(* IEC 61131-3 sources: learning-path/05_oop_in_st/exercises/2_interfaces/src, 2 files *)

(* ---- basicTank.st ---- *)
NAMESPACE FluidHandlingClass

    //Update the class to implement the Interface
    class Tank
        VAR PUBLIC
            inletValve: ValveClass;
            outletValve: ValveClass;
        END_VAR

        METHOD PRIVATE OpenInlet
            inletValve.Open();
        END_METHOD
        METHOD PRIVATE OpenOutlet
            outletValve.Open();
        END_METHOD
        METHOD PRIVATE CloseInlet
            inletValve.Close();
        END_METHOD
        METHOD PRIVATE CloseOutlet
            outletValve.Close();
        END_METHOD

        METHOD PUBLIC Fill
            this.OpenInlet();
            this.CloseOutlet();
        END_METHOD

        METHOD PUBLIC Flush
            this.OpenInlet();
            this.OpenOutlet();
        END_METHOD

        METHOD PUBLIC Close
            this.CloseInlet();
            this.CloseOutlet();
        END_METHOD

        METHOD PUBLIC Emptying
            this.CloseInlet();
            this.OpenOutlet();
        END_METHOD
    END_CLASS
END_NAMESPACE

(* ---- basicValve.st ---- *)
NAMESPACE FluidHandlingClass
    CLASS basicValve
        VAR
            _ctrlOpen : BOOL;
            _state : ValveState;
            _isClosed : BOOL;
            _isOpen : BOOL;
        END_VAR

        METHOD PUBLIC Open
            _ctrlOpen := TRUE;
            _isOpen := TRUE;
            _isClosed := FALSE;
        END_METHOD

        METHOD PUBLIC Close
            _ctrlOpen := FALSE;
            _isOpen := FALSE;
            _isClosed := TRUE;
        END_METHOD

        METHOD PUBLIC GetState: FluidHandlingClass.ValveState
            IF (_ctrlOpen) THEN
                GetState := ValveState#Open;
            ELSE
                GetState := ValveState#Closed;
            END_IF;
            _state := GetState;
        END_METHOD

        METHOD PUBLIC WriteCyclic
            VAR_OUTPUT
                ctrlOpen : BOOL;
                isOpen : BOOL;
                isClosed : BOOL;
                state : ValveState;
            END_VAR
            ctrlOpen := _ctrlOpen;
            isOpen := _isOpen;
            isClosed := _isClosed;
            state := _state;
        END_METHOD
    END_CLASS
END_NAMESPACE
